// TIA Portal V19 export
TYPE "LAF_typeNgConveyorEm1ParametersInterface"
// stored: Access Published
   STRUCT
      configuration : "LAF_typeNgConveyorEm1Parameters";
      commands : "LBC_typeInterfaceCommands";
      monitoring { S7_SetPoint := 'True'} : "LAF_typeNgConveyorEm1ProcessValues";
   END_STRUCT;
END_TYPE
